// TIA Portal V18 export
DATA_BLOCK "Function_Selection_HMI"   // DB278
{ S7_Optimized_Access := 'TRUE' }
VERSION : 0.1
// stored: AutoNumber true, DBAccessibleFromOPCUA true, IsOnlyStoredInLoadMemory false, IsRetainMemResEnabled false, IsWriteProtectedInAS false, MemoryReserve 100
   VAR
      "Deaering A" : Bool;
      "Deaering B" : Bool;
      "Recirculation A" : Bool;
      "Recirculation B" : Bool;
      Recirculation : Bool;
      "Pressure release A" : Bool;
      "Pressure release B" : Bool;
      "Pressure release" : Bool;
      "Dearing A Without valve" : Bool;
      "Dearing B Without valve" : Bool;
      "Shot metering" : Bool;
      "Continuous metering" : Bool;
      "Metering program" : Bool;
      "Pre run" : Bool;
      "ratio check" : Bool;
      Flush : Bool;
   END_VAR
   VAR RETAIN
      SnuffBack : Bool;
      SnunfBack_flow : Real;
      Snuffback_qty : Real;
   END_VAR
   VAR
      Function_Snuffback_volume_dispensed : Real;
      "Condition Check A" : Bool;
      "Condition Check B" : Bool;
      "Snuffback selected" : Bool;
      "Snuffback start" : Bool;
   END_VAR
BEGIN
END_DATA_BLOCK
